# EPICS substitutions: ioc/PSCApp/Db/out_register.substitutions
file db/out_register.db {
    pattern {OUT_REGISTER_NUMBER}
        {"1"}
}
